# EPICS substitutions: apps/mpodLvApp/Db/fttrklv.substitutions
file "db/mpod8008l.db" {
    pattern {HOST,CH,SCAN,PORT,DETALIAS}
{"129.57.86.97","0","2 second","B_HW_FTTLV_Sl0_Ch0","B_DET_FTT_LV_0"}
{"129.57.86.97","1","2 second","B_HW_FTTLV_Sl0_Ch1","B_DET_FTT_LV_1"}
}
